TYPE EL3052_PDOS :
	STRUCT
		
		HwToPLC : EL3052_HWTOPLC_PDOS;
		
	END_STRUCT
END_TYPE

(* stored: Version 1.1.0.1, ProductVersion 3.1.4024.15
   DUT EL3052_PDOS: Id {db49b0ea-39ce-417b-adb0-40098b614258} *)
